(*
 * Contains every service relevant to Resi4MPM control.
 * Used so that the services can use each other (similar to dependency injection).
 *)
FUNCTION_BLOCK ServiceContainer
VAR_INPUT
END_VAR
VAR_OUTPUT
END_VAR
VAR
	m_ptrGvlInterface: POINTER TO GvlInterfaceBase;
	m_ptrErrorMgr: POINTER TO ErrorManagerBase;
	
	m_pm: ProcessManager;
	m_ptrProcessManager: POINTER TO ProcessManager := ADR(m_pm);
 
	m_st: StateTracker;
	m_ptrStateTracker: POINTER TO StateTracker := ADR(m_st);

	m_rc: RaConnector;
	m_ptrRaConnector: POINTER TO RaConnector := ADR(m_rc);
END_VAR

METHOD FB_init : BOOL
VAR_INPUT
	bInitRetains : BOOL; // if TRUE, the retain variables are initialized (warm start / cold start)
	bInCopyCode : BOOL;  // if TRUE, the instance afterwards gets moved into the copy code (online change)
	
	i_ptrGvlInterface: POINTER TO GvlInterfaceBase;
	i_ptrErrorMgr: POINTER TO ErrorManagerBase;
END_VAR
// get the APPLICATION-SPECIFIC services
THIS^.m_ptrGvlInterface := i_ptrGvlInterface;
THIS^.m_ptrErrorMgr := i_ptrErrorMgr;

// initialize all services
THIS^.m_ptrProcessManager^.ProvideServices(THIS^.m_ptrStateTracker, THIS^.m_ptrRaConnector);
THIS^.m_ptrRaConnector^.ProvideServices(THIS^.m_ptrGvlInterface, THIS^.m_ptrProcessManager, THIS^.m_ptrStateTracker, THIS^.m_ptrErrorMgr);
THIS^.m_ptrStateTracker^.ProvideServices(THIS^.m_ptrProcessManager, THIS^.m_ptrRaConnector);
END_METHOD

PROPERTY PtrGvlInterface : POINTER TO GvlInterfaceBase
GET
PtrGvlInterface := THIS^.m_ptrGvlInterface;
END_GET
END_PROPERTY

PROPERTY PtrProcessManager : POINTER TO ProcessManager
GET
PtrProcessManager := THIS^.m_ptrProcessManager;
END_GET
END_PROPERTY

PROPERTY PtrRaConnector : POINTER TO RaConnector
GET
PtrRaConnector := THIS^.m_ptrRaConnector;
END_GET
END_PROPERTY

PROPERTY PtrStateTracker : POINTER TO StateTracker
GET
PtrStateTracker := THIS^.m_ptrStateTracker;
END_GET
END_PROPERTY

END_FUNCTION_BLOCK

(* stored: Version 1.1.0.1, ProductVersion 3.1.4024.9
   POU ServiceContainer: Id {55cc9c46-6acb-446f-9720-88ef800cc500}, SpecialFunc None
   Method FB_init: Id {19a79c36-0ca7-4778-ba5c-dff66cd4ee09}
   Property PtrGvlInterface: Id {82d5ee62-b111-4d29-9dd5-cc3f3f660dc9}
   Get Get: Id {fade7e1e-0009-49c7-81d3-2055004d188a}
   Property PtrProcessManager: Id {6ea69623-d10c-4741-846e-84eb12aced5e}
   Get Get: Id {0d76a124-1ba9-4eba-9803-c11e3c654886}
   Property PtrRaConnector: Id {fb4b3f3d-0b0d-49ea-be34-884ec953a250}
   Get Get: Id {99fe007b-7882-4f4d-a183-c40ec8d0c0d6}
   Property PtrStateTracker: Id {c3b894aa-cdfd-4649-a8b1-770eaccbea44}
   Get Get: Id {199d3f36-fe48-4a9d-8aed-8201584481cf} *)
